{attribute 'qualified_only'}
{attribute 'hide'}
VAR_GLOBAL CONSTANT
	kMaxCount : UDINT := 100;
	kName : STRING := 'app';
END_VAR

(* stored: Version 1.1.0.1
   GVL GParams: Id {g} *)
